FUNCTION_BLOCK FB_Solenoid EXTENDS FB_Device
VAR_INPUT
	bNormallyOpen:BOOL;//True if Valve is Normally Open
	bCmdOpen:BOOL;// True if Valve should be opened
END_VAR
VAR
	bTheoreticallyOpen:BOOL;//Internal variable to control state of the valve, true when valve is open
END_VAR
VAR_OUTPUT
	bCoilEnergiseState:BOOL;//Signal sent to coil to energise
	eSolenoidState: E_SolenoidState;//If coil is not energised in reality
END_VAR

//Call method open or close depending on command to valve
IF bCmdOpen THEN
	M_Open();
ELSE
    M_Close();
END_IF

METHOD M_CheckState
//Return the state enum of the valve 
IF bTheoreticallyOpen THEN
	eSolenoidState := E_SolenoidState.Open;
ELSE
	eSolenoidState := E_SolenoidState.Closed;
END_IF
END_METHOD

METHOD PUBLIC M_Close
//Call base M_Cyclic logic from FB_Device
hr:=SUPER^.M_CyclicLogic();
//Close the valve if the device is enabled
IF bDeviceEnable THEN
	IF bNormallyOpen THEN
		bCoilEnergiseState := TRUE;
		bTheoreticallyOpen := FALSE;
	ELSE
		bCoilEnergiseState := FALSE;
		bTheoreticallyOpen := bNormallyOpen;
	END_IF
ELSE
	bCoilEnergiseState := FALSE;
	bTheoreticallyOpen := bNormallyOpen;
END_IF
M_CheckState();
END_METHOD

METHOD PUBLIC M_Open
////Call base M_Cyclic logic from FB_Device
hr:=SUPER^.M_CyclicLogic();
//Open the valve if the device is enabled
IF bDeviceEnable THEN
	IF NOT bNormallyOpen THEN
		bCoilEnergiseState := TRUE;
		bTheoreticallyOpen := TRUE;
	ELSE
		bCoilEnergiseState := FALSE;
		bTheoreticallyOpen := bNormallyOpen;
	END_IF
ELSE
	bCoilEnergiseState := FALSE;
	bTheoreticallyOpen := bNormallyOpen;
END_IF
M_Checkstate();
END_METHOD

END_FUNCTION_BLOCK

(* stored: Version 1.1.0.1
   POU FB_Solenoid: Id {a7e2e3b9-dfd6-4640-b79e-2b5bc5bc4dd9}, SpecialFunc None
   Method M_CheckState: Id {876197d4-1678-4755-bfce-9f51e76cf52b}
   Method M_Close: Id {9936ae59-63a8-4842-acb7-0972cbd832e2}
   Method M_Open: Id {e0f7a43f-bf45-4aad-b570-5a1a3b451270} *)
